(* IEC 61131-3 sources: IecStringProject/_internal/release/IecFrmtStr/V0.02.0, 1 file *)

(* ---- IecFrmtStr.fun ---- *)
FUNCTION fnIecFormatString : UDINT
	VAR_INPUT
		pDestination : UDINT;
		DestinationLength : UDINT;
		pSource : UDINT;
		pArguments : UDINT;
	END_VAR
END_FUNCTION
